FUNCTION Camera_Set_Int : Buffer_Error
VAR_INPUT
	Camera : REFERENCE TO Cognex_Camera;
	Num : USINT;
	In : INT;
END_VAR

Camera_Set_Int := Set_Int_From_Buffer(	In:= In, 
										Num:= Num, 
										Layout:= Camera.Ouput_Buffer_Layout, 
										Buffer:= Camera.User_Data.UserData);

END_FUNCTION

(* stored: Version 1.1.0.1, ProductVersion 3.1.4024.10
   POU Camera_Set_Int: Id {127b00c9-8357-4eae-abf6-0d3b388870df}, SpecialFunc None *)
